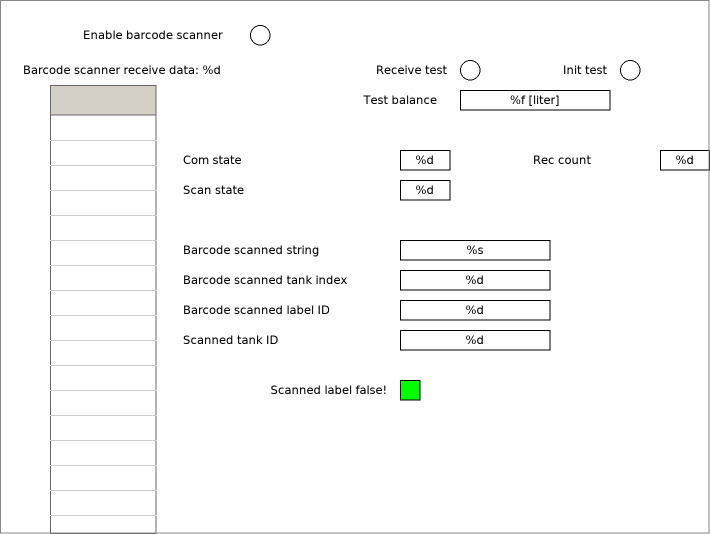
VISUALIZATION VISU_BARCODE  // 710x534
    Table (50,85 106x449), data array: PRG_INK.cI_Barcode_RxBuff
        p2232123230: PRG_INK.cI_Barcode_RxBuff[INDEX]
        p511219082: PRG_PRINT.sL_SensorResults[INDEX].yMark
        p1755163831: PRG_PRINT.sL_SensorResults[INDEX].phiMark
        p4092479075: PRG_PRINT.sL_SensorResults[INDEX].xCam
        p2237128397: PRG_PRINT.sL_SensorResults[INDEX].yCam
        p505689113: PRG_PRINT.sL_SensorResults[INDEX].phiCam
        p1757482276: PRG_PRINT.sL_SensorResults[INDEX].dx
        p4088588272: PRG_PRINT.sL_SensorResults[INDEX].dy
        p2243050616: PRG_PRINT.sL_SensorResults[INDEX].dphi
    Rectangle (20,60 240x20), "Barcode scanner receive data: %d", text variable: PRG_INK.iI_Barcode_RecDataLength
    Rectangle (400,240 150x20), "%s", text variable: PRG_INK.fb_BarcodeStoragetank.aL_ReceivedData
    Rectangle (180,240 200x20), "Barcode scanned string"
    Rectangle (400,270 150x20), "%d", text variable: PRG_INK.fb_BarcodeStoragetank.iL_ScannedStorageIndex
    Rectangle (180,270 200x20), "Barcode scanned tank index"
    Rectangle (400,300 150x20), "%d", text variable: PRG_INK.fb_BarcodeStoragetank.lL_ScannedLabel
    Rectangle (180,300 200x20), "Barcode scanned label ID"
    Rectangle (400,330 150x20), "%d", text variable: PRG_INK.sAdsIkInkStorageTank[PRG_INK.fb_BarcodeStoragetank.iL_ScannedStorageIndex].sI_InkParameter.iScannerId
        OnMouseClick: write the text variable via Default
    Rectangle (180,330 200x20), "Scanned tank ID"
    Rectangle (219,380 171x20), "Scanned label false!"
    RoundedRectangle (400,380 20x20), colour toggle: PRG_INK.fb_BarcodeStoragetank.bO_LabelScanFalse[PRG_INK.fb_BarcodeStoragetank.iL_ScannedStorageIndex]
    Rectangle (80,25 160x20), "Enable barcode scanner"
    Ellipse (250,25 20x20), colour toggle: PRG_INK.bI_EnableBarcodeScanner
        toggle PRG_INK.bI_EnableBarcodeScanner
    Rectangle (355,60 95x20), "Receive test"
    Ellipse (460,60 20x20), colour toggle: PRG_INK.bI_Barcode_DataRec
        tap PRG_INK.bI_Barcode_DataRec
    Rectangle (400,180 50x20), "%d", text variable: PRG_INK.fb_BarcodeStoragetank.iL_ScanState
        OnMouseClick: write the text variable via Default
    Rectangle (180,180 200x20), "Scan state"
    Rectangle (515,60 95x20), "Init test"
    Ellipse (620,60 20x20), colour toggle: PRG_INK.bI_Barcode_AckInit
        tap PRG_INK.bI_Barcode_AckInit
    Rectangle (400,150 50x20), "%d", text variable: PRG_INK.fb_BarcodeStoragetank.iL_COMstate
        OnMouseClick: write the text variable via Default
    Rectangle (180,150 200x20), "Com state"
    Rectangle (460,90 150x20), "%f [liter]", text variable: PRG_INK.FB_BalanceLink.fO_Readings[PRG_INK.fb_BarcodeStoragetank.iL_ScannedStorageIndex]
        OnMouseClick: write the text variable via Default
    Rectangle (329,90 111x20), "Test balance"
    Rectangle (660,150 50x20), "%d", text variable: PRG_INK.fb_BarcodeStoragetank.iL_ReceiveCount
    Rectangle (530,150 102x20), "Rec count"
END_VISUALIZATION

(* stored: Version 1.1.0.1, ProductVersion 3.1.4024.9
   Visu VISU_BARCODE: Id {99c1f80b-6031-4242-9e14-df8f000ff086} *)
